(* PLC project Unnamed, Unknown Unnamed 1 *)
(* stored: creationDateTime 2026-05-15T20:13:33, modificationDateTime 2026-05-15T20:13:33 *)

PROGRAM main
  VAR
    Green : BOOL := FALSE;
    Yellow : BOOL := FALSE;
    Red : BOOL := FALSE;
    GreenOn : BOOL := True;
    YellowOn : BOOL := False;
    RedOn : BOOL := False;
    GreenTimer : TON;
    YellowTimer : TON;
    RedTimer : TON;
  END_VAR

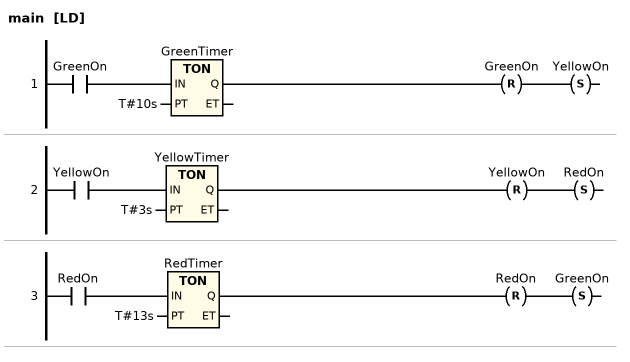
(* LD diagram, written out as Structured Text *)
GreenTimer(IN := GreenOn, PT := T#10s);
IF GreenTimer.Q THEN GreenOn := FALSE; END_IF;
IF GreenTimer.Q THEN YellowOn := TRUE; END_IF;
YellowTimer(IN := YellowOn, PT := T#3s);
IF YellowTimer.Q THEN YellowOn := FALSE; END_IF;
IF YellowTimer.Q THEN RedOn := TRUE; END_IF;
RedTimer(IN := RedOn, PT := T#13s);
IF RedTimer.Q THEN RedOn := FALSE; END_IF;
IF RedTimer.Q THEN GreenOn := TRUE; END_IF;
END_PROGRAM

CONFIGURATION Config0
  RESOURCE Res0 ON PLC
    TASK task0(INTERVAL := T#20ms, PRIORITY := 1);
    PROGRAM instance0 WITH task0 : main;
  END_RESOURCE
END_CONFIGURATION
